// TIA Portal V20 export
DATA_BLOCK "InstGetIdentMv"   // DB220
// stored: InstanceOfName GetIdentMv, InstanceOfType FB
"GetIdentMv"
   // VAR_INPUT
   //    identMvAllUnits { ExternalAccessible := 'False'; ExternalVisible := 'False'; ExternalWritable := 'False'} : Array[1.."NO_OF_UNITS"] of "typeEMIdentMv";
   //    numberOfMvReaders : USInt;
   // END_VAR
   // VAR_OUTPUT
   //    selectedUnit : USInt;
   //    selectedEM : USInt;
   //    error : Word;
   // END_VAR
   // VAR_IN_OUT
   //    IdentMvInterfaceHmi : "typeIdentMvHmi";
   // END_VAR
   // VAR
   //    statSelectedEMIdentMv : USInt;
   //    statSelectedUnitIdentRMv : USInt;
   // END_VAR
BEGIN
END_DATA_BLOCK
